Yaskawa INFORM job: PICK.JBI

/JOB
//NAME PICK
//POS
///NPOS 0,0,0,2,0,0
///USER 9
///TOOL 0
///POSTYPE USER
///RECTAN
///RCONF 0,0,0,0,0,0,0,0
P084=0.000,0.000,-35.000,0.00,0.00,0.00
P085=0.000,0.000,35.000,0.00,0.00,0.00
//INST
///DATE 2018/02/02 16:57
///COMM OPDR1
///ATTR SC,RW
///GROUP1 RB1
NOP
DOUT OG#(1) 1
'gripper open
TIMER T=0.50
IMOV P084 V=100.0 PL=0 UF#(9)
'naar beneden
DOUT OG#(1) 2
'gripper dicht
TIMER T=0.50
IMOV P085 V=100.0 PL=0 UF#(9)
'naar boven
END
